// TwinCAT 3 PLC project PalettenstationPLC
// ProgramVersion: 3.1.4024.0
// libraries:
//   Tc2_Standard, * (Beckhoff Automation GmbH)
//   Tc2_System, * (Beckhoff Automation GmbH)
//   Tc3_Module, * (Beckhoff Automation GmbH)
// project tree:
//   GVLs/ GVL_IO.TcGVL, GVL_Simulation.TcGVL
//   / PlcTask.TcTTO
//   POUs/ MAIN.TcPOU
// real-time tasks:
//   TASK PlcTask: cycle T#10ms, priority 20, ADS port 350
// I/O:
//   DEVICE Gerät 1 (EtherCAT), AmsNetId 5.35.203.54.2.1
//     Klemme 1 (EK1100) [EK1100 EtherCAT-Koppler (2A E-Bus)]
//       Klemme 2 (EL1002) [EL1002 2K. Dig. Eingang 24V, 3ms]
//       Klemme 3 (EL1004) [EL1004 4K. Dig. Eingang 24V, 3ms]
//       Klemme 4 (EL1004) [EL1004 4K. Dig. Eingang 24V, 3ms]
//       Klemme 5 (EL1008) [EL1008 8K. Dig. Eingang 24V, 3ms]
//       Klemme 6 (EL2004) [EL2004 4K. Dig. Ausgang 24V, 0.5A]
//       Klemme 7 (EL2004) [EL2004 4K. Dig. Ausgang 24V, 0.5A]
//       Klemme 8 (EL2008) [EL2008 8K. Dig. Ausgang 24V, 0.5A]
//       Klemme 9 (EL3064) [EL3064 4K.Ana. Eingang 0-10V]
//       Klemme 10 (EL3144) [EL3144 4K. Ana. Eingang 0-20mA]
//       Klemme 11 (EL3204) [EL3204 4K. Ana. Eingang PT100 (RTD)]
//       Klemme 12 (EL4014) [EL4014 4K. Ana. Ausgang 0-20mA, 12bit]
//       Klemme 13 (EK1110) [EK1110 EtherCAT-Verlängerung]
// variable links:
//   PalettenstationPLC/PalettenstationPLC Instance <-> Device 1 (EtherCAT)/Term 1 (EK1100)/Term 2 (EL1002)
//     PlcTask Inputs/GVL_IO.DI_NotHaltFrei <-> Channel 2/Input

CONFIGURATION PalettenstationPLC
    RESOURCE PLC ON TwinCAT3
        TASK PlcTask(INTERVAL := T#10ms, PRIORITY := 20);
        PROGRAM MAIN WITH PlcTask : MAIN;
    END_RESOURCE
END_CONFIGURATION

// ---- GVLs/GVL_IO.TcGVL
{attribute 'qualified_only'}
VAR_GLOBAL

    // ==================================================
    // DIGITALE EINGÄNGE
    // ==================================================

    DI_NotHaltFrei        AT %I* : BOOL;
    DI_SchutzhaubeZu      AT %I* : BOOL;
    DI_PaletteEingang     AT %I* : BOOL;
    DI_PalettePositioniert AT %I* : BOOL;
    DI_HubUnten           AT %I* : BOOL;
    DI_HubOben            AT %I* : BOOL;
    DI_KollisionFrei      AT %I* : BOOL;
    DI_WerkerQuittierung  AT %I* : BOOL;


    // ==================================================
    // DIGITALE AUSGÄNGE
    // ==================================================

    DO_SignalGruen        AT %Q* : BOOL;
    DO_AlarmRot           AT %Q* : BOOL;
    DO_Foerderband        AT %Q* : BOOL;
    DO_FoerderbandStopp   AT %Q* : BOOL;
    DO_HubwerkHoch        AT %Q* : BOOL;
    DO_HubwerkRunter      AT %Q* : BOOL;
    DO_ProzessFreigabe    AT %Q* : BOOL;
    DO_Heizfreigabe       AT %Q* : BOOL;


    // ==================================================
    // ANALOGE EINGÄNGE
    // ==================================================

    AI_FolienTemperatur   AT %I* : REAL;
    AI_MotorTemperatur    AT %I* : REAL;

	// ==================================================
	// INTERNE PROGRAMMVARIABLEN
	// ==================================================
	
	Schritt : INT := 0;
	AlarmAktiv : BOOL := FALSE;


END_VAR

// ---- GVLs/GVL_Simulation.TcGVL
{attribute 'qualified_only'}
VAR_GLOBAL
	SIM_NotHaltFrei         : BOOL := TRUE;
    SIM_SchutzhaubeZu       : BOOL := TRUE;
    SIM_PaletteEingang      : BOOL := FALSE;
    SIM_PalettePositioniert : BOOL := FALSE;
    SIM_HubUnten            : BOOL := TRUE;
    SIM_HubOben             : BOOL := FALSE;
    SIM_KollisionFrei       : BOOL := TRUE;
    SIM_WerkerQuittierung   : BOOL := FALSE;
END_VAR

// ---- POUs/MAIN.TcPOU
PROGRAM MAIN
VAR
	tProzesszeit : TON;
	
	bNotHaltFrei         : BOOL;
    bSchutzhaubeZu       : BOOL;
    bPaletteEingang      : BOOL;
    bPalettePositioniert : BOOL;
    bHubUnten            : BOOL;
    bHubOben             : BOOL;
    bKollisionFrei       : BOOL;
    bWerkerQuittierung   : BOOL;
	
END_VAR

// =====================================================
// AUSGÄNGE ZU BEGINN JEDES SPS-ZYKLUS ZURÜCKSETZEN
// =====================================================

GVL_IO.DO_SignalGruen      := FALSE;
GVL_IO.DO_AlarmRot         := FALSE;
GVL_IO.DO_Foerderband      := FALSE;
GVL_IO.DO_FoerderbandStopp := FALSE;
GVL_IO.DO_HubwerkHoch      := FALSE;
GVL_IO.DO_HubwerkRunter    := FALSE;
GVL_IO.DO_ProzessFreigabe  := FALSE;
GVL_IO.DO_Heizfreigabe     := FALSE;


// VAR ... END_VAR
// Die Reihenfolge ist damit 
//→ Umschaltung Simulation/Hardware
// → CASE-Struktur

// lesen -->  Programm ausführen -->  E/A schreiben --> wieder von vorne
// =====================================================
// SCHRITTKETTE
// =====================================================

CASE GVL_IO.Schritt OF

    0:// S0 - Anlage bereit und wartet auf Palette

        GVL_IO.DO_SignalGruen := TRUE;

        IF GVL_IO.DI_NotHaltFrei
           AND GVL_IO.DI_SchutzhaubeZu
           AND GVL_IO.DI_HubUnten
           AND GVL_IO.DI_PaletteEingang THEN

            GVL_IO.Schritt := 1;

        END_IF


    1: // S1 - Förderband transportiert Palette

        GVL_IO.DO_Foerderband := TRUE;

        IF NOT GVL_IO.DI_NotHaltFrei THEN

            GVL_IO.Schritt := 8;

        ELSIF GVL_IO.DI_PalettePositioniert THEN

            GVL_IO.Schritt := 2;

        END_IF


    2: // S2 - Palette stoppen

        GVL_IO.DO_FoerderbandStopp := TRUE;

        // Im nächsten SPS-Zyklus zu Hubwerk hoch
        GVL_IO.Schritt := 3;


    3: // S3 - Hubwerk fährt nach oben

        GVL_IO.DO_FoerderbandStopp := TRUE;
        GVL_IO.DO_HubwerkHoch      := TRUE;

        IF NOT GVL_IO.DI_NotHaltFrei
           OR NOT GVL_IO.DI_KollisionFrei THEN

            GVL_IO.Schritt := 8;

        ELSIF GVL_IO.DI_HubOben THEN

            GVL_IO.Schritt := 4;

        END_IF


    4: // S4 - Temperatur prüfen

        GVL_IO.DO_FoerderbandStopp := TRUE;
        GVL_IO.DO_Heizfreigabe     := TRUE;

        IF GVL_IO.AI_MotorTemperatur > 100.0 THEN

            GVL_IO.Schritt := 8;

        ELSIF GVL_IO.AI_FolienTemperatur >= 165.0
           AND GVL_IO.AI_FolienTemperatur <= 185.0 THEN

            GVL_IO.Schritt := 5;

        ELSE

            GVL_IO.Schritt := 8;

        END_IF


    5: // S5 - Bearbeitung läuft fünf Sekunden

        GVL_IO.DO_FoerderbandStopp := TRUE;
        GVL_IO.DO_Heizfreigabe     := TRUE;
        GVL_IO.DO_ProzessFreigabe  := TRUE;

        tProzesszeit(
            IN := TRUE,
            PT := T#5S
        );

        IF GVL_IO.AI_FolienTemperatur < 165.0
           OR GVL_IO.AI_FolienTemperatur > 185.0
           OR GVL_IO.AI_MotorTemperatur > 100.0
           OR NOT GVL_IO.DI_NotHaltFrei THEN

            tProzesszeit(IN := FALSE);
            GVL_IO.Schritt := 8;

        ELSIF tProzesszeit.Q THEN

            tProzesszeit(IN := FALSE);
            GVL_IO.Schritt := 6;

        END_IF


    6: // S6 - Hubwerk fährt nach unten

        GVL_IO.DO_FoerderbandStopp := TRUE;
        GVL_IO.DO_HubwerkRunter    := TRUE;

        IF NOT GVL_IO.DI_NotHaltFrei THEN

            GVL_IO.Schritt := 8;

        ELSIF GVL_IO.DI_HubUnten THEN

            GVL_IO.Schritt := 7;

        END_IF


    7: // S7 - Palette verlässt Station

        GVL_IO.DO_Foerderband := TRUE;

        IF NOT GVL_IO.DI_PalettePositioniert THEN

            GVL_IO.Schritt := 0;

        END_IF


    8: // S8 - Alarm setzen

        GVL_IO.AlarmAktiv := TRUE;
        GVL_IO.Schritt := 9;


    9: // S9 - Warten auf Fehlerbeseitigung und Quittierung

        GVL_IO.DO_AlarmRot := TRUE;

        IF GVL_IO.DI_WerkerQuittierung
           AND GVL_IO.DI_NotHaltFrei
           AND GVL_IO.AI_FolienTemperatur >= 165.0
           AND GVL_IO.AI_FolienTemperatur <= 185.0
           AND GVL_IO.AI_MotorTemperatur <= 100.0 THEN

            GVL_IO.AlarmAktiv := FALSE;
            GVL_IO.Schritt := 0;

        END_IF


    ELSE // Unbekannter Schrittwert

        GVL_IO.AlarmAktiv := TRUE;
        GVL_IO.Schritt := 9;

END_CASE

END_PROGRAM
